{attribute 'linkalways'} 
{attribute 'no_explicit_call' := 'This FB is a CLASS and must be accessed using methods or properties'}
{attribute 'enable_dynamic_creation'}
FUNCTION_BLOCK Queue EXTENDS Disposable IMPLEMENTS I_Queue
VAR
	linkedList : LinkedList;
	eventEmitter : EventEmitter;
END_VAR

METHOD PUBLIC AddItem
VAR_INPUT
	Item : ANY;
END_VAR
Enqueue(Item);
END_METHOD

METHOD PUBLIC Clear
linkedList.Clear();
EmitChangedEvent();
END_METHOD

METHOD PUBLIC Contains : BOOL;
VAR_INPUT
	Item : ANY;
END_VAR
VAR
	found : I_LinkedListNode;
END_VAR
found := linkedList.Find(Item);
Contains := found <> 0;
END_METHOD

PROPERTY PUBLIC Count : DINT
GET
Count := linkedList.Count;
END_GET
END_PROPERTY

METHOD PRIVATE EmitChangedEvent
VAR
	pCollectionChangedEvent : POINTER TO CollectionChangedEvent;
END_VAR
pCollectionChangedEvent := __NEW(CollectionChangedEvent(Target := THIS^));
eventEmitter.Emit('OnChanged', pCollectionChangedEvent^);
pCollectionChangedEvent^.Dispose();
END_METHOD

METHOD PRIVATE EmitDisposedEvent
VAR
	pCollectionDisposedEvent : POINTER TO CollectionDisposedEvent;
END_VAR
pCollectionDisposedEvent := __NEW(CollectionDisposedEvent(Target := THIS^));
eventEmitter.Emit('OnDisposed', pCollectionDisposedEvent^);
pCollectionDisposedEvent^.Dispose();
END_METHOD

METHOD PUBLIC Enqueue
VAR_INPUT
	Item : ANY;
END_VAR
linkedList.AddLast(Item);
EmitChangedEvent();
END_METHOD

METHOD FB_exit : BOOL
VAR_INPUT
	bInCopyCode : BOOL; // if TRUE, the exit method is called for exiting an instance that is copied afterwards (online change).
END_VAR
IF bInCopyCode THEN
	RETURN;
END_IF

Clear();
EmitDisposedEvent();
END_METHOD

METHOD PUBLIC GetEnumerator : I_ForwardEnumerator
GetEnumerator := linkedList.GetEnumerator();
END_METHOD

PROPERTY IsEmpty : BOOL
GET
IsEmpty := linkedList.IsEmpty;
END_GET
END_PROPERTY

METHOD PUBLIC OffEvent
VAR_INPUT
	EventName : T_MaxString;
	EventHandler : I_EventHandler;
END_VAR
eventEmitter.OffEvent(EventName, EventHandler);
END_METHOD

METHOD PUBLIC OnceEvent
VAR_INPUT
	EventName : T_MaxString;
	EventHandler : I_EventHandler;
END_VAR
eventEmitter.OnceEvent(EventName, EventHandler);
END_METHOD

METHOD PUBLIC OnEvent
VAR_INPUT
	EventName : T_MaxString;
	EventHandler : I_EventHandler;
END_VAR
eventEmitter.OnEvent(EventName, EventHandler);
END_METHOD

METHOD PUBLIC TryCopyTo : BOOL
VAR_INPUT
	Destination : ANY;
END_VAR
TryCopyTo := linkedList.TryCopyTo(Destination);
END_METHOD

METHOD PUBLIC TryCopyToLocation : BOOL
VAR_INPUT
	DestinationAddress : PVOID;
	DestinationSize : UDINT;
END_VAR
TryCopyToLocation := linkedList.TryCopyToLocation(DestinationAddress, DestinationSize);
END_METHOD

METHOD PUBLIC TryDequeue : BOOL;
VAR_INPUT
	Destination : ANY;
END_VAR
VAR
	first : I_LinkedListNode;
	dequeued : BOOL;
END_VAR
first := linkedList.First;

IF first = 0 THEN
	RETURN;
END_IF

dequeued := linkedList.First.TryGet(Destination);

IF NOT dequeued THEN
	RETURN;
END_IF

linkedList.RemoveFirst();
EmitChangedEvent();
TryDequeue := TRUE;
END_METHOD

METHOD PUBLIC TryPeek : BOOL;
VAR_INPUT
	Destination : ANY;
END_VAR
VAR
	first : I_LinkedListNode;
END_VAR
first := linkedList.First;

IF first = 0 THEN
	RETURN;
END_IF

TryPeek := first.TryGet(Destination);
END_METHOD

METHOD PUBLIC TryRemoveItem : BOOL
VAR_INPUT
	Item : ANY;
END_VAR
TryRemoveItem := linkedList.TryRemoveItem(Item);
EmitChangedEvent();
END_METHOD

END_FUNCTION_BLOCK

(* stored: Version 1.1.0.1, ProductVersion 3.1.4024.12
   POU Queue: Id {f74e450d-364c-02f8-170a-18b41d891a1b}, SpecialFunc None
   Folder Destructor: Id {f5924f56-29c7-030a-30f3-14b75bebc4cd}
   Folder Private: Id {e8aa5d0f-f71d-00df-20e8-9b69262afc14}
   Method AddItem: Id {c77a3bb0-c156-0de4-15eb-bdeeda91fe2f}
   Method Clear: Id {29186540-cdf0-011d-3459-08f489335b10}
   Method Contains: Id {d68f157a-0e90-0e8f-2c39-73e1da0acfad}
   Property Count: Id {32ffea39-9406-042e-333c-0accc5dd1865}
   Get Get: Id {ad6373c7-15aa-0106-31aa-5e0d07edf6b4}
   Method EmitChangedEvent: Id {2c23aad8-f5d9-02f8-0a89-777afd4371e1}
   Method EmitDisposedEvent: Id {c08f0b80-4b01-0b65-35e8-3483823483b6}
   Method Enqueue: Id {c2b816e4-7255-0e77-373d-b08574d12c41}
   Method FB_exit: Id {ec600dee-d548-0cfa-1aef-c150514e6db9}
   Method GetEnumerator: Id {a671f2aa-d11c-0752-2b3d-c25ded0c0fd6}
   Property IsEmpty: Id {3ea718af-156f-0220-23dd-af1b15ca28c0}
   Get Get: Id {d92a4d3a-198b-03a2-1821-8b552e2e6731}
   Method OffEvent: Id {bbfef87e-f191-0255-2771-deb965bf2ea0}
   Method OnceEvent: Id {e4f10eb2-7d73-09d6-0c0c-9faf9d2a3f5e}
   Method OnEvent: Id {34e9c52b-20b4-06c3-20b0-24e332ea2ecf}
   Method TryCopyTo: Id {4d3ff1aa-2a63-0ec2-0445-407d6d12688d}
   Method TryCopyToLocation: Id {578a15c7-1b6b-018b-0f83-00a1c4ac9041}
   Method TryDequeue: Id {fd5964c6-9076-0deb-1c39-dcdacc888477}
   Method TryPeek: Id {546650f0-772d-06b9-3312-e9757a915b5b}
   Method TryRemoveItem: Id {1a15878f-9053-0e32-21d0-b0e6ff65bc75} *)
